Staubli VAL3: F6_testmove.pgx

program F6_testmove()
  local num l_ni
  local bool l_bTemp
  local joint l_jTemp1
  local num l_nCount
begin
  //call FC_InitMotion()
  if bTxtPrSv==false
    popUpMsg("请首先对点位文件初始化（按F3-PoIn）")
  else
    pointToJoint(tTool,jConfig,pfrmCad[0],jConfig)
    MoveTo.trsf=pfrmCad[0].trsf
    l_bTemp=pointToJoint(tTool,jConfig,MoveTo,l_jTemp1)
    movej(l_jTemp1,tTool,mNomSpeed)
    l_nCount=0
    do
      if pfrmCad[l_nCount].trsf!={0,0,0,0,0,0}
        /////运动部分/////
        MoveTo.trsf=pfrmCad[l_nCount].trsf
        l_bTemp=pointToJoint(tTool,jConfig,MoveTo,l_jTemp1)
        movej(l_jTemp1,tTool,mNomSpeed)
        delay(0)
        /////运动部分/////
        pfrmCad[l_nCount].trsf={0,0,0,0,0,0}
        if l_nCount==600
          bTxt1=true
        endIf
        if l_nCount==1100
          bTxt2=true
        endIf
        if l_nCount==100
          bTxt3=true
        endIf
      endIf
      if l_nCount==1499
        l_nCount=0
      else
        l_nCount=l_nCount+1
      endIf
      delay(0)
    until pfrmCad[l_nCount].trsf=={0,0,0,0,0,0}
    bTxtPrSv=false
  endIf
  sScrPts="NotReady"
  call hmi_refreshmain()
  //
  //
  waitEndMove()
  popUpMsg("test over")
  //call FC_EndMotion()
end
